TEXTLIST EL1904_M_1
  1 = 'Emergency Stop A' | chinese: '急停A' | Chinese: '急停A'
  2 = 'Emergency Stop B' | chinese: '急停B' | Chinese: '急停B'
  3 = 'Fast Scan left limit' | chinese: 'Fast Scan 左极限' | Chinese: 'Fast Scan 左极限'
  4 = 'Fast Scan right limit' | chinese: 'Fast Scan 右极限' | Chinese: 'Fast Scan 右极限'
   = ''
END_TEXTLIST

(* stored: Version 1.1.0.1, ProductVersion 3.1.4024.11
   TextList EL1904_M_1: Id {dad84e2f-f2f2-403f-a5e3-2e585d2c4cbc} *)
